(* PLC project Unnamed, Unknown Unnamed 1 *)
(* stored: creationDateTime 2022-08-16T15:49:17, modificationDateTime 2024-11-22T10:55:53 *)

PROGRAM main
  VAR
    TOF0 : TOF;
    TON0 : TON;
  END_VAR
  VAR
    blink_led0 AT %QX0.0 : BOOL;
    blink_led1 AT %QX0.1 : BOOL;
    blink_led2 AT %QX6.3 : BOOL;
  END_VAR
  VAR
    blink_led3 : BOOL;
  END_VAR
  VAR
    blink_led4 AT %QX0.4 : BOOL;
    blink_led5 AT %QX0.5 : BOOL;
    blink_led6 AT %QX0.6 : BOOL;
    blink_led7 AT %QX0.7 : BOOL;
    Analog_A0 AT %IW0 : INT;
    Analog_A1 AT %IW1 : INT;
    Analog_A2 AT %IW2 : INT;
    Analog_A3 AT %IW3 : INT;
  END_VAR
  VAR
    Analog_A0_value : INT;
    Analog_A1_value : INT;
    Analog_A2_value : INT;
    Analog_A3_value : INT;
  END_VAR

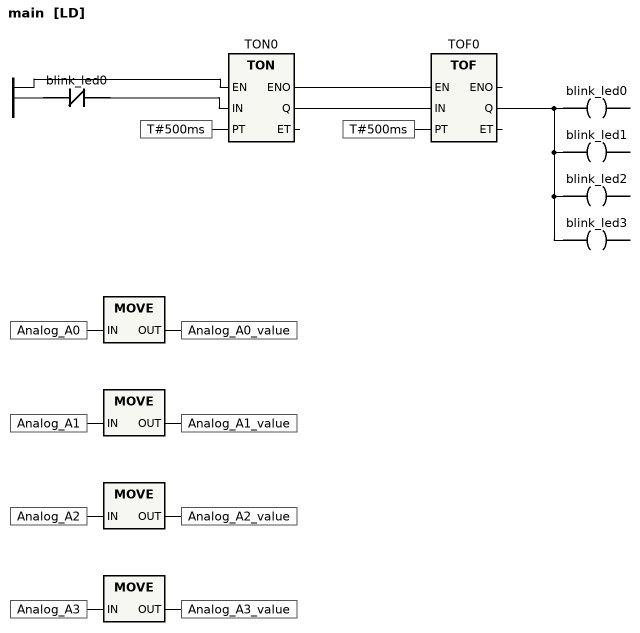
(* LD diagram, written out as Structured Text *)
TON0(IN := NOT blink_led0, PT := T#500ms);
TOF0(EN := TON0.ENO, IN := TON0.Q, PT := T#500ms);
blink_led0 := TOF0.Q;
Analog_A0_value := Analog_A0;
Analog_A1_value := Analog_A1;
Analog_A2_value := Analog_A2;
Analog_A3_value := Analog_A3;
blink_led1 := TOF0.Q;
blink_led2 := TOF0.Q;
blink_led3 := TOF0.Q;
END_PROGRAM

PROGRAM kiban_hanso
  VAR
    ita_hanso_start : BOOL;
    ita_hanso_il : BOOL;
    ita_hanso_running : BOOL;
    ita_hanso_B0 : BOOL;
    ita_hanso_B1 : BOOL;
    ita_hanso_B2 : BOOL;
    ita_hanso_B3 : BOOL;
  END_VAR
  VAR
    Sensor_fiber1 AT %IX0.0 : BOOL;
    Sensor_fiber2 AT %IX0.1 : BOOL;
    Sensor_metal AT %IX0.2 : BOOL;
  END_VAR
  VAR
    ita_kakunin_ok : BOOL;
    TON0 : TON;
    TON1 : TON;
    kiban_nai_ERR : BOOL;
  END_VAR
  VAR_EXTERNAL
    position_motor1_1 : DWORD;
    position_motor2_1 : DWORD;
  END_VAR
  VAR
    idou_pos_hansou AT %MD0 : DWORD := 30000;
    idou_pos_pickup AT %MD1 : DWORD := 30000;
  END_VAR
  VAR
    en_motor1 : BOOL;
  END_VAR
  VAR_EXTERNAL
    cw_m1 : BOOL;
    ccw_m1 : BOOL;
  END_VAR
  VAR
    ccw_m1_on : BOOL;
    cw_m1_on : BOOL;
  END_VAR
  VAR_EXTERNAL
    data_moto1 : BYTE;
    data_moto2 : BYTE;
    current_M1_pos : DWORD;
    current_M2_pos : DWORD;
  END_VAR
  VAR
    current_1_vitri : DWORD;
  END_VAR
  VAR_EXTERNAL
    motor1_speed : UINT;
    motor2_speed : UINT;
  END_VAR
  VAR
    set_motor1_speed : UINT;
    set_motor1_accel : UINT;
  END_VAR
  VAR_EXTERNAL
    motor1_accel : UINT;
    motor2_accel : UINT;
  END_VAR
  VAR
    mode_run_m1 : BYTE;
  END_VAR
  VAR_EXTERNAL
    START_Moto_1 : BOOL;
    START_Moto_2 : BOOL;
    motor1_running : BOOL;
    motor1_position_ok : BOOL;
    motor2_position_ok : BOOL;
    zero_m1_kaki_ok : BOOL;
    lr_0 : BOOL;
    lr_1 : BOOL;
    lr_2 : BOOL;
    lr_3 : BOOL;
    dm_0 : DWORD;
    dm_1 : DWORD;
    dm_2 : DWORD;
    dm_3 : DWORD;
    dm_4 : DWORD;
  END_VAR
  VAR
    dm_input0 : DWORD;
    dm_input1 : DWORD;
    dm_input2 : DWORD;
    dm_input3 : DWORD;
    dm_input4 : DWORD;
    kb_hansou_idouOK : BOOL;
    pickup_idouOK : BOOL;
    pickup_siji : BOOL;
    save0 : BOOL;
    save1 : BOOL;
    save2 : BOOL;
    save3 : BOOL;
    save4 : BOOL;
  END_VAR
  VAR  (* added by the conversion: wires and edge detectors of the diagram *)
    _MOVE39_ENO : BOOL;
    _MOVE39_OUT : DWORD;
    _EQ67_ENO : BOOL;
    _EQ67_OUT : BOOL;
    _MOVE25_ENO : BOOL;
    _MOVE25_OUT : DWORD;
    _EQ43_ENO : BOOL;
    _EQ43_OUT : BOOL;
  END_VAR

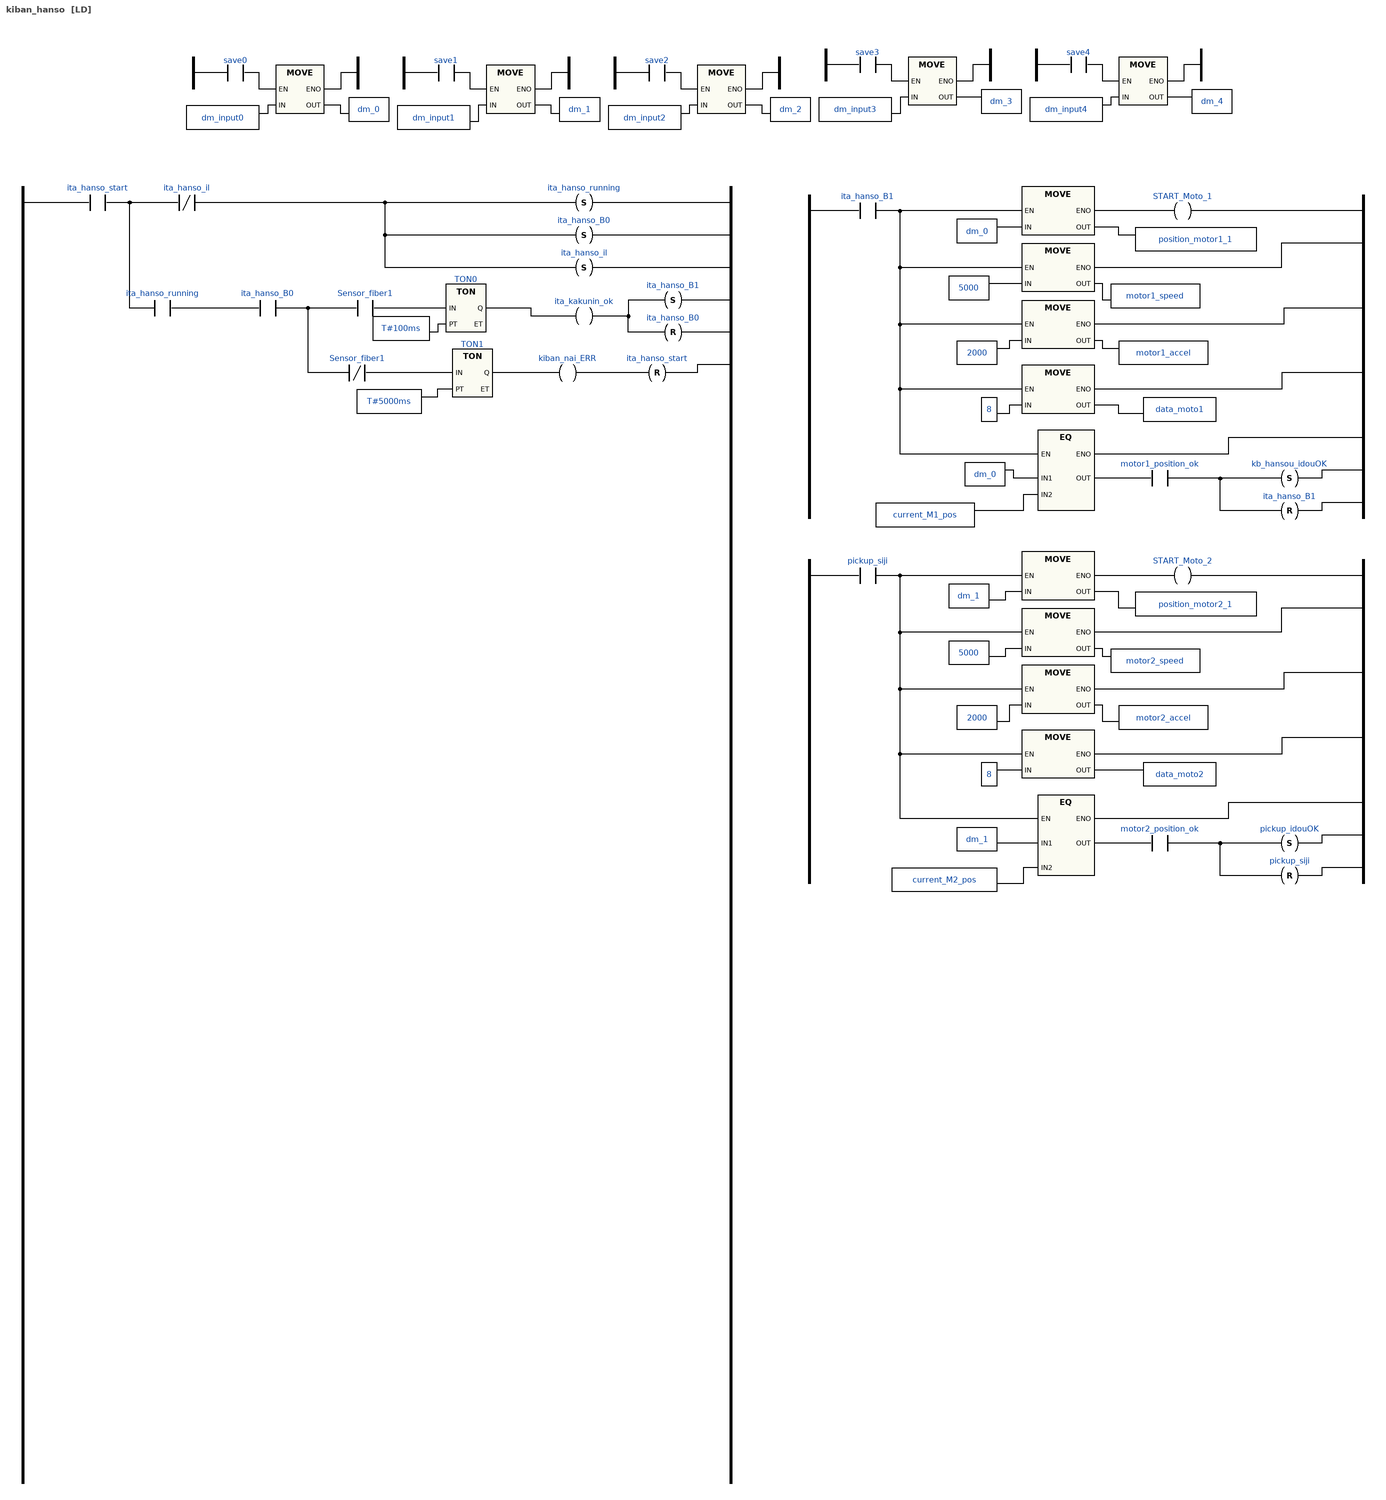
(* LD diagram, written out as Structured Text *)
IF ita_hanso_start AND NOT ita_hanso_il THEN ita_hanso_running := TRUE; END_IF;
IF ita_hanso_start AND NOT ita_hanso_il THEN ita_hanso_B0 := TRUE; END_IF;
IF ita_hanso_start AND NOT ita_hanso_il THEN ita_hanso_il := TRUE; END_IF;
TON0(IN := ita_hanso_start AND ita_hanso_running AND ita_hanso_B0 AND Sensor_fiber1, PT := T#100ms);
ita_kakunin_ok := TON0.Q;
TON1(IN := ita_hanso_start AND ita_hanso_running AND ita_hanso_B0 AND NOT Sensor_fiber1, PT := T#5000ms);
kiban_nai_ERR := TON1.Q;
IF TON0.Q THEN ita_hanso_B1 := TRUE; END_IF;
IF TON0.Q THEN ita_hanso_B0 := FALSE; END_IF;
IF TON1.Q THEN ita_hanso_start := FALSE; END_IF;
_MOVE39_OUT := MOVE(EN := ita_hanso_B1, IN := dm_0, ENO => _MOVE39_ENO);
START_Moto_1 := _MOVE39_ENO;
IF _MOVE39_ENO THEN position_motor1_1 := _MOVE39_OUT; END_IF;
IF ita_hanso_B1 THEN motor1_speed := 5000; END_IF;
IF ita_hanso_B1 THEN motor1_accel := 2000; END_IF;
IF ita_hanso_B1 THEN data_moto1 := 8; END_IF;
_EQ67_OUT := EQ(EN := ita_hanso_B1, IN1 := dm_0, IN2 := current_M1_pos, ENO => _EQ67_ENO);
IF _EQ67_OUT AND motor1_position_ok THEN ita_hanso_B1 := FALSE; END_IF;
IF _EQ67_OUT AND motor1_position_ok THEN kb_hansou_idouOK := TRUE; END_IF;
_MOVE25_OUT := MOVE(EN := pickup_siji, IN := dm_1, ENO => _MOVE25_ENO);
START_Moto_2 := _MOVE25_ENO;
IF _MOVE25_ENO THEN position_motor2_1 := _MOVE25_OUT; END_IF;
IF pickup_siji THEN motor2_speed := 5000; END_IF;
IF pickup_siji THEN motor2_accel := 2000; END_IF;
IF pickup_siji THEN data_moto2 := 8; END_IF;
_EQ43_OUT := EQ(EN := pickup_siji, IN1 := dm_1, IN2 := current_M2_pos, ENO => _EQ43_ENO);
IF _EQ43_OUT AND motor2_position_ok THEN pickup_siji := FALSE; END_IF;
IF _EQ43_OUT AND motor2_position_ok THEN pickup_idouOK := TRUE; END_IF;
IF save0 THEN dm_0 := dm_input0; END_IF;
IF save1 THEN dm_1 := dm_input1; END_IF;
IF save2 THEN dm_2 := dm_input2; END_IF;
IF save3 THEN dm_3 := dm_input3; END_IF;
IF save4 THEN dm_4 := dm_input4; END_IF;
END_PROGRAM

CONFIGURATION Config0
  RESOURCE Res0 ON PLC
    TASK task0(INTERVAL := T#5ms, PRIORITY := 0);
    TASK task1(INTERVAL := T#10ms, PRIORITY := 0);
    PROGRAM instance1 WITH task0 : main;
    PROGRAM instance2 WITH task1 : kiban_hanso;
  END_RESOURCE
END_CONFIGURATION
